// TIA Portal V19 export
DATA_BLOCK "IN"   // DB28
{ S7_Optimized_Access := 'FALSE' }
   VAR
      EMG_STOP : Bool;
      HOOTER_RESET : Bool;
      POWER_FAIL : Bool;
      "PUMP-1_TRIP" : Bool;
      "PUMP-2_TRIP" : Bool;
      SWT_LL : Bool;
      SWT_ML : Bool;
      SWT_HL : Bool;
      PWT_LL : Bool;
      PWT_ML : Bool;
      PWT_HL : Bool;
      ALKALI_LL : Bool;
      ALAKLI_HL : Bool;
      ACID_LL : Bool;
      ACID_HL : Bool;
      LSW_FWD_PUMP : Bool;
      LSW_RET_PUMP : Bool;
      AIR_SWITCH : Bool;
      CT_SENSOR : Int;
      PH_SENSOR : Int;
      TEMP_SENSOR : Int;
   END_VAR
BEGIN
END_DATA_BLOCK
